FUNCTION_BLOCK FB_BaseRecipe_HMI EXTENDS FB_Base IMPLEMENTS ITF_BaseRecipe_HMI
VAR
	itfBaseRecipe			: ITF_BaseRecipe_HMI_Connector;
	refstRepiceData			: REFERENCE TO ST_BaseRecipe_HMI;
	
END_VAR

(*			
	RafalOS
	Rafał Osajda		03.03.2025		TC 4026.13		wer. 0.0.0.1
	Kopiuje składniki z wybranej receptury i tworzy nową recepture
*)
METHOD PUBLIC AddRecipeFromRecipe : BOOL
VAR_INPUT
	uiNumberRecipe				: UINT;
	stTexts						: ST_BaseLabel;
END_VAR
THIS^.itfBaseRecipe.AddRecipeFromRecipe (
	uiNumberRecipe 	:= uiNumberRecipe,
	stTexts			:= stTexts
);
END_METHOD

(*			
	RafalOS
	Rafał Osajda		03.03.2025		TC 4026.13		wer. 0.0.0.1
	Kopiuje składniki z wybranego szablonu i tworzy nową recepture
*)
METHOD PUBLIC AddRecipeFromTemplate : BOOL
VAR_INPUT
	uiNumberTemplates			: UINT;
	stTexts						: ST_BaseLabel;
END_VAR
THIS^.itfBaseRecipe.AddRecipeFromTemplate (
	uiNumberTemplates 	:= uiNumberTemplates,
	stTexts				:= stTexts
);
END_METHOD

(*			
	RafalOS
	Rafał Osajda		25.10.2025		TC 4024.66
	Utworzenie nowych szablonów receptur na podstawie dodanych fb zewnętrznych - wywołanie metody powoduje
	skosowanie dotychczasowych szablonów i receptur
*)
METHOD PUBLIC CreateRecipeTemplates : BOOL
VAR_INPUT
END_VAR
THIS^.itfBaseRecipe.CreateTemplates ();
END_METHOD

(*			
	RafalOS
	Rafał Osajda		03.03.2025		TC 4026.13		wer. 0.0.0.1
	
*)
METHOD PUBLIC DeleteRecipe : BOOL
VAR_INPUT
	uiNumber				: uint;
END_VAR
THIS^.itfBaseRecipe.DeleteRecipe (uiNumber := uiNumber);
END_METHOD

METHOD FB_init : BOOL
VAR_INPUT
	bInitRetains : BOOL; // if TRUE, the retain variables are initialized (warm start / cold start)
	bInCopyCode : BOOL;  // if TRUE, the instance afterwards gets moved into the copy code (online change)
	fbBaseRecipe			: ITF_BaseRecipe_HMI_Connector;
END_VAR
THIS^.itfBaseRecipe := fbBaseRecipe;
END_METHOD

(*			
	RafalOS
	Rafał Osajda		03.03.2025		TC 4026.13		wer. 0.0.0.1
	
*)
METHOD PUBLIC GetIngredientFromRecipe : ST_BaseDescriptor
VAR_INPUT
	uiNumberOfRecipe			: UINT;
	uiNumberOfIngredient		: UINT;
END_VAR
GetIngredientFromRecipe			:= THIS^.itfBaseRecipe.GetIngredientFromRecipe (
									uiNumberOfRecipe := uiNumberOfRecipe,
									uiNumberOfIngredient := uiNumberOfIngredient
								);
END_METHOD

(*			
	RafalOS
	Rafał Osajda		02.12.2025		TC 4024.66
	Zwraca do tablicy wybrany zakres składników
*)
METHOD PUBLIC GetIngredientRange 
VAR_INPUT
	iRecipe			: INT;	//numer receptury z której bierzemy składniki
	iStartIndex		: INT;	//numer startowy składnika
	iCount			: INT;	//ilośc pobieranych 
END_VAR
VAR_IN_OUT
	arrOut : ARRAY [*] OF ST_BaseDescriptor;
END_VAR
VAR_OUTPUT
	iNumberOfFilledData	: INT;	//ilosc wypelnionych danych na strone
END_VAR
THIS^.itfBaseRecipe.GetIngredientRange (
	iRecipe		:= iRecipe,
	iStartIndex	:= iStartIndex,
	iCount		:= iCount,
	arrOut		:= arrOut,
	iNumberOfFilledData	=> iNumberOfFilledData
);
END_METHOD

METHOD GetNameList : ST_BaseRecipeList
VAR_INPUT
END_VAR
GetNameList := THIS^.itfBaseRecipe.GetNameList ();
END_METHOD

METHOD GetNameListTemplate : ST_BaseRecipeList
VAR_INPUT
END_VAR
GetNameListTemplate := THIS^.itfBaseRecipe.GetNameListTemplate ();
END_METHOD

(*			
	RafalOS
	Rafał Osajda		03.03.2025		TC 4026.13		wer. 0.0.0.1
	
*)
METHOD PUBLIC GetNumberIngredientOfRecipe : UINT
VAR_INPUT
	uiNumber				: UINT;
END_VAR
GetNumberIngredientOfRecipe 		:= THIS^.itfBaseRecipe.GetNumberIngredientOfRecipe (uiNumber := uiNumber);
END_METHOD

METHOD PUBLIC GetNumberOfRecipe : UINT
VAR_INPUT
END_VAR
GetNumberOfRecipe			:= THIS^.itfBaseRecipe.GetNumberOfRecipe ();
END_METHOD

METHOD PUBLIC GetNumberOfTemplate : UINT
VAR_INPUT
END_VAR
GetNumberOfTemplate		:= THIS^.itfBaseRecipe.GetNumberOfTemplate ();
END_METHOD

METHOD PUBLIC LinkRecipeDataHMI : BOOL
VAR_INPUT
	stRecipe			: REFERENCE TO ST_BaseRecipe_HMI;
END_VAR
THIS^.refstRepiceData REF= stRecipe;
END_METHOD

END_FUNCTION_BLOCK

(* stored: Version 1.1.0.1
   POU FB_BaseRecipe_HMI: Id {bad54886-8f7a-0ae3-3994-568964574923}, SpecialFunc None
   Folder WiazanieZmiennych: Id {2049a495-6e2a-073c-3f15-28145b6ad20f}
   Method AddRecipeFromRecipe: Id {aae3ed58-2935-02d5-0d7e-f8f398061af9}
   Method AddRecipeFromTemplate: Id {01a5fe38-bdca-05d8-3e4b-ba9cac535b5e}
   Method CreateRecipeTemplates: Id {26a4ef2c-be17-02db-05eb-ccea8127fa7c}
   Method DeleteRecipe: Id {00f6da5c-db94-013f-2d96-a723e24f04b4}
   Method FB_init: Id {c599964b-6b59-014c-0aad-068a83dd644f}
   Method GetIngredientFromRecipe: Id {7a734e23-0984-074b-2673-48b478218584}
   Method GetIngredientRange: Id {6a211e5e-6d99-0aed-03e6-91d1253a40d5}
   Method GetNameList: Id {f870dd41-4bca-0468-2631-2fd1688facf9}
   Method GetNameListTemplate: Id {d8e956a5-eae8-0659-13a8-d001e5530f78}
   Method GetNumberIngredientOfRecipe: Id {583ae13c-d0e1-0a7d-356b-82e75f1a3572}
   Method GetNumberOfRecipe: Id {891c6672-0914-06c5-3261-b421315a92a6}
   Method GetNumberOfTemplate: Id {4b01afa7-0b73-02ee-189b-e8ad25b9b9f4}
   Method LinkRecipeDataHMI: Id {ac4eb793-b833-00fc-3c7b-28667d82ba04} *)
